FUNCTION_BLOCK KeepCurrentOpCdtLogic (* Composite Function Block Type *)
  (* Standard: 61499-2 *)
  (* Version 0.0, 8/20/2024, SESA713705, Schneider Electric, template *)
  PACKAGE SE.Nereda;
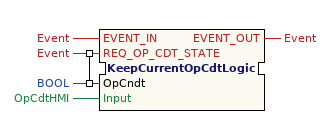
  EVENT_INPUT
    EVENT_IN; (* Initialization Request *)
    REQ_OP_CDT_STATE WITH OpCndt; (* Normal Execution Request *)
  END_EVENT
  EVENT_OUTPUT
    EVENT_OUT; (* Initialization Confirm *)
  END_EVENT
  VAR_INPUT
    OpCndt : BOOL;
  END_VAR
  SOCKETS
    Input : OpCdtHMI;
  END_SOCKETS
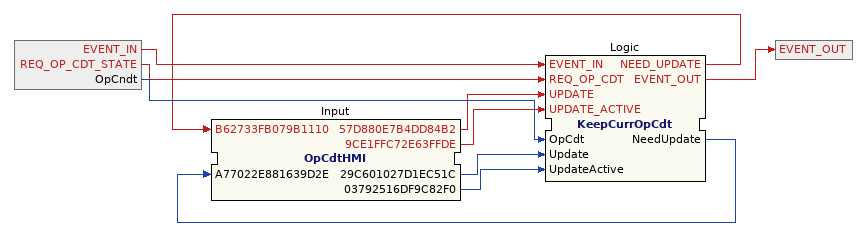
  FBS
    Logic : KeepCurrOpCdt;
  END_FBS
  EVENT_CONNECTIONS
    EVENT_IN TO Logic.EVENT_IN;
    REQ_OP_CDT_STATE TO Logic.REQ_OP_CDT;
    Input.57D880E7B4DD84B2 TO Logic.UPDATE;
    Input.9CE1FFC72E63FFDE TO Logic.UPDATE_ACTIVE;
    Logic.NEED_UPDATE TO Input.B62733FB079B1110;
    Logic.EVENT_OUT TO EVENT_OUT;
  END_CONNECTIONS
  DATA_CONNECTIONS
    OpCndt TO Logic.OpCdt;
    Input.29C601027D1EC51C TO Logic.Update;
    Input.03792516DF9C82F0 TO Logic.UpdateActive;
    Logic.NeedUpdate TO Input.A77022E881639D2E;
  END_CONNECTIONS
END_FUNCTION_BLOCK
